// TIA Portal V19 export
TYPE "LAF_typeAxisDiagData"
TITLE = LAF_typeAxisDiagData
// Diagnostic information of a Technology Object
// stored: Access Published
   STRUCT
      "type" { ExternalWritable := 'False'} : UDInt;   // Type of axis (0=no axis, 1=speed axis, 2=positioning axis, 3=synchronous axis, 4=external encoder)
      values { ExternalWritable := 'False'} : "LAF_typeAxisDiagValues";
      statusAxis { ExternalWritable := 'False'} : "LAF_typeAxisDiagStatus";
      statusSensor { ExternalWritable := 'False'} : "LAF_typeAxisDiagStatusSensor";
      statusPositioning { ExternalWritable := 'False'} : "LAF_typeAxisDiagStatusPositioning";
      units { ExternalWritable := 'False'} : "LAF_typeAxisDiagUnits";
   END_STRUCT;
END_TYPE
